PROGRAM MAIN
VAR

	Timer : LREAL;
	

	
END_VAR

//Timer
Timer := Timer + 0.001;

ActuationSystems();
P_Joy();

END_PROGRAM

(* stored: Version 1.1.0.1, ProductVersion 3.1.4024.9
   POU MAIN: Id {d1c7ef4e-0337-49c7-9736-af80a39f1b25}, SpecialFunc None *)
